(* CODESYS project czas_reakcji.project

Project tree, tasks and I/O mapping:
  Device : CODESYS Control Win V3, 3S - Smart Software Solutions GmbH, order no. 305021, version 3.5.8.10
    application Application
      libraries: Standard, * (System)
      task MainTask (cyclic, interval t#20ms, priority 1) calls PLC_PRG
      task VISU_TASK (cyclic, interval 100 ms, priority 31) calls VisuElems.Visu_Prg
      program PLC_PRG [ST]
      visualisation Visualization
  text list GlobalTextList
*)

// Device/Application/PLC_PRG
PROGRAM PLC_PRG
VAR
	_TIME: TON;
	COUNTER : CTU;
	
	TIMER : TON;
	LIGHTER : CTU;

	DELAY : TON;
	DELAYER : CTU;
	
	BTN_1 : BOOL;
	BTN_2 : BOOL;
	BTN_3 : BOOL;
	BTN_4 : BOOL;
	
	IS_CLICKED_1 : BOOL;
	IS_CLICKED_2 : BOOL;
	IS_CLICKED_3 : BOOL;
	IS_CLICKED_4 : BOOL;
	
	LAMP_1 : BOOL;
	LAMP_2 : BOOL;
	LAMP_3 : BOOL;
	LAMP_4 : BOOL;
	
	COME_IN: BOOL := TRUE;
	
	SCORE: WORD := 0;
	PROBE: WORD := 0;
	
END_VAR

_TIME(PT:=T#1MS, IN := NOT _TIME.Q);
COUNTER(CU:=_TIME.Q, RESET:=COUNTER.Q, PV:=15);



IF COME_IN THEN
	IF COUNTER.CV >= 0 AND COUNTER.CV <= 3 THEN
		_TIME.IN := FALSE;
		COME_IN := FALSE;
	
		LAMP_1 := TRUE;
		LAMP_2 := FALSE;
		LAMP_3 := FALSE;
		LAMP_4 := FALSE;
		COME_IN := FALSE;
		
		TIMER(PT:=T#1MS, IN := NOT TIMER.Q);
		LIGHTER(CU:=TIMER.Q, RESET:=FALSE, PV:=705);
		IF LIGHTER.CV > 200 THEN
			LAMP_1 := FALSE;
		END_IF
		
		IF LIGHTER.CV > 200 AND BTN_1 THEN
			SCORE := SCORE +1;
		END_IF
		
		IF LIGHTER.CV > 700 THEN
			_TIME.IN := NOT _TIME.Q;
			COME_IN := TRUE;
			PROBE := PROBE +1;
		END_IF
	ELSIF COUNTER.CV > 3 AND COUNTER.CV <= 7 THEN
		_TIME.IN := FALSE;
		COME_IN := FALSE;
		
		LAMP_1 := FALSE;
		LAMP_2 := TRUE;
		LAMP_3 := FALSE;
		LAMP_4 := FALSE;
		COME_IN := FALSE;
		
		TIMER(PT:=T#1MS, IN := NOT TIMER.Q);
		LIGHTER(CU:=TIMER.Q, RESET:=FALSE, PV:=705);
		IF LIGHTER.CV > 200 THEN
			LAMP_1 := FALSE;
		END_IF
		
		IF LIGHTER.CV > 200 AND BTN_1 THEN
			SCORE := SCORE +1;
		END_IF
		
		IF LIGHTER.CV > 700 THEN
			_TIME.IN := NOT _TIME.Q;
			COME_IN := TRUE;
			PROBE := PROBE +1;
		END_IF
	ELSIF COUNTER.CV > 7 AND COUNTER.CV <= 12 THEN
		_TIME.IN := FALSE;
		COME_IN := FALSE;
		
		LAMP_1 := FALSE;
		LAMP_2 := FALSE;
		LAMP_3 := TRUE;
		LAMP_4 := FALSE;
		COME_IN := FALSE;
		
		TIMER(PT:=T#1MS, IN := NOT TIMER.Q);
		LIGHTER(CU:=TIMER.Q, RESET:=FALSE, PV:=705);
		IF LIGHTER.CV > 200 THEN
			LAMP_1 := FALSE;
		END_IF
		
		IF LIGHTER.CV > 200 AND BTN_1 THEN
			SCORE := SCORE +1;
		END_IF
		
		IF LIGHTER.CV > 700 THEN
			_TIME.IN := NOT _TIME.Q;
			COME_IN := TRUE;
			PROBE := PROBE +1;
		END_IF
	ELSE
		_TIME.IN := FALSE;
		COME_IN := FALSE;
		
		LAMP_1 := FALSE;
		LAMP_2 := FALSE;
		LAMP_3 := FALSE;
		LAMP_4 := TRUE;
		COME_IN := FALSE;
		
		TIMER(PT:=T#1MS, IN := NOT TIMER.Q);
		LIGHTER(CU:=TIMER.Q, RESET:=FALSE, PV:=705);
		IF LIGHTER.CV > 200 THEN
			LAMP_1 := FALSE;
		END_IF
		
		IF LIGHTER.CV > 200 AND BTN_1 THEN
			SCORE := SCORE +1;
		END_IF
		
		IF LIGHTER.CV > 700 THEN
			_TIME.IN := NOT _TIME.Q;
			COME_IN := TRUE;
			PROBE := PROBE +1;
		END_IF
	END_IF
END_IF

IF PROBE = 15 THEN
	COME_IN := FALSE;
	_TIME.IN := FALSE;
	TIMER.IN := FALSE;
	
	DELAY(PT:=T#10MS, IN := NOT DELAY.Q);
	DELAYER(CU:=DELAY.Q, RESET:=FALSE, PV:=500);
	
	CASE PROBE OF
	1: 
		LAMP_1 := FALSE;  //0
		LAMP_2 := FALSE;  //0
		LAMP_3 := FALSE;  //0
		LAMP_4 := TRUE;   //1
	2: 
		LAMP_1 := FALSE;  //0
		LAMP_2 := FALSE;  //0
		LAMP_3 := TRUE;   //1
		LAMP_4 := FALSE;  //0
	3: 
		LAMP_1 := FALSE;  //0
		LAMP_2 := FALSE;  //0
		LAMP_3 := TRUE;   //1
		LAMP_4 := TRUE;   //1
	4: 
		LAMP_1 := FALSE;  //0
		LAMP_2 := TRUE;   //1
		LAMP_3 := FALSE;  //0
		LAMP_4 := FALSE;  //0
	5: 
		LAMP_1 := FALSE;  //0
		LAMP_2 := TRUE;   //1
		LAMP_3 := FALSE;  //0
		LAMP_4 := TRUE;   //1
	6: 
		LAMP_1 := FALSE;  //0
		LAMP_2 := TRUE;   //1
		LAMP_3 := TRUE;   //1
		LAMP_4 := FALSE;  //0
	7: 
		LAMP_1 := FALSE;  //0
		LAMP_2 := TRUE;   //1
		LAMP_3 := TRUE;   //1
		LAMP_4 := TRUE;   //1
	8: 
		LAMP_1 := TRUE;   //1
		LAMP_2 := FALSE;  //0
		LAMP_3 := FALSE;  //0
		LAMP_4 := FALSE;  //0
	9: 
		LAMP_1 := TRUE;   //1
		LAMP_2 := FALSE;  //0
		LAMP_3 := FALSE;  //0
		LAMP_4 := TRUE;   //1
	10: 
		LAMP_1 := TRUE;   //1
		LAMP_2 := FALSE;  //0
		LAMP_3 := TRUE;   //1
		LAMP_4 := FALSE;  //0
	11: 
		LAMP_1 := TRUE;   //1
		LAMP_2 := FALSE;  //0
		LAMP_3 := TRUE;   //1
		LAMP_4 := TRUE;   //1
	12: 
		LAMP_1 := TRUE;   //1
		LAMP_2 := TRUE;   //1
		LAMP_3 := FALSE;  //0
		LAMP_4 := FALSE;  //0
	13: 
		LAMP_1 := TRUE;   //1
		LAMP_2 := TRUE;   //1
		LAMP_3 := FALSE;  //0
		LAMP_4 := TRUE;   //1
	14: 
		LAMP_1 := TRUE;   //1
		LAMP_2 := TRUE;   //1
		LAMP_3 := TRUE;   //1
		LAMP_4 := FALSE;  //0
	15: 
		LAMP_1 := TRUE;   //1
		LAMP_2 := TRUE;   //1
		LAMP_3 := TRUE;   //1
		LAMP_4 := TRUE;   //1
	ELSE
		LAMP_1 := FALSE;  //0
		LAMP_2 := FALSE;  //0
		LAMP_3 := FALSE;  //0
		LAMP_4 := FALSE;  //0		
	END_CASE
END_IF

END_PROGRAM

// Device/Application/Visualization
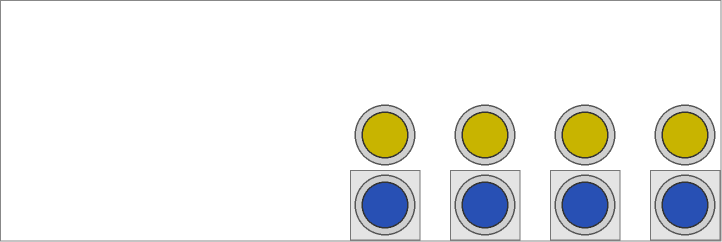
VISUALIZATION Visualization  // 722x242
    Lamp1 (350,100 70x70), variable: PLC_PRG.LAMP_1, style: Lamp-Lamp1-Yellow
    Lamp1 (450,100 70x70), variable: PLC_PRG.LAMP_2, style: Lamp-Lamp1-Yellow
    Lamp1 (550,100 70x70), variable: PLC_PRG.LAMP_3, style: Lamp-Lamp1-Yellow
    Lamp1 (650,100 70x70), variable: PLC_PRG.LAMP_4, style: Lamp-Lamp1-Yellow
    PushSwitch (350,170 70x70), variable: PLC_PRG.BTN_1, behaviour: TAP, style: Switch-PushSwitch-Blue
    PushSwitch (450,170 70x70), variable: PLC_PRG.BTN_2, behaviour: TAP, style: Switch-PushSwitch-Blue
    PushSwitch (550,170 70x70), variable: PLC_PRG.BTN_3, behaviour: TAP, style: Switch-PushSwitch-Blue
    PushSwitch (650,170 70x70), variable: PLC_PRG.BTN_4, behaviour: TAP, style: Switch-PushSwitch-Blue
END_VISUALIZATION
